Fanuc KAREL source: libmathex.kl

-- Copyright (c) 2016, G.A. vd. Hoorn
--
-- Licensed under the Apache License, Version 2.0 (the "License");
-- you may not use this file except in compliance with the License.
-- You may obtain a copy of the License at
--
--     http://www.apache.org/licenses/LICENSE-2.0
--
-- Unless required by applicable law or agreed to in writing, software
-- distributed under the License is distributed on an "AS IS" BASIS,
-- WITHOUT WARRANTIES OR CONDITIONS OF ANY KIND, either express or implied.
-- See the License for the specific language governing permissions and
-- limitations under the License.


PROGRAM libmathex
--------------------------------------------------------------------------------
--
-- libmathex implementation
--
-- author: G.A. vd. Hoorn
--
--------------------------------------------------------------------------------
%ALPHABETIZE
%COMMENT = 'ROS//r0'
%NOBUSYLAMP
%NOLOCKGROUP
%NOPAUSE = COMMAND + TPENABLE + ERROR




--------------------------------------------------------------------------------
--
-- local types & constants
--
--------------------------------------------------------------------------------




--------------------------------------------------------------------------------
--
-- remote routine prototypes
--
--------------------------------------------------------------------------------




--------------------------------------------------------------------------------
--
-- local routine prototypes
--
--------------------------------------------------------------------------------
%INCLUDE mathex\mathex.klh




--------------------------------------------------------------------------------
--
-- Empty body
--
--------------------------------------------------------------------------------
BEGIN
END libmathex




ROUTINE signi
BEGIN
	IF (val = 0) THEN RETURN (0); ENDIF
	RETURN (val DIV (ABS(val)))
END signi




ROUTINE signr
BEGIN
	IF (val > 0.0) THEN RETURN ( 1.0); ENDIF
	IF (val < 0.0) THEN RETURN (-1.0); ENDIF
	RETURN (0.0)
END signr
